TYPE LinearPositions :
STRUCT
	deployed	:LREAL:=500;
	stowed		:LREAL:=100;
	maintenance	:LREAL:=0;	

END_STRUCT
END_TYPE

(* stored: Version 1.1.0.1, ProductVersion 3.1.4024.12
   DUT LinearPositions: Id {6f796ba7-fc5e-4ff1-a527-119668af3216} *)
